(* IEC 61131-3 sources: plc_on_fpga_riscv_hybrid/RV_FPGA_PLC_IDE_Projects/Or, 1 file *)

(* ---- Or.il ---- *)
VAR
END_VAR

PROGRAM Or
    R1 :
        LD     %KEY.0
        OR     %KEY.1
        ST     %LEDG.0
END_PROGRAM
